TYPE ST_HMI_SAFETY_IN :
STRUCT
	bQuitSafety,
	
	bQuitAreaST10,
	bUnlockDoorST33	: BOOL;
END_STRUCT
END_TYPE

(* stored: Version 1.1.0.1, ProductVersion 3.1.4024.12
   DUT ST_HMI_SAFETY_IN: Id {ab1ef7de-b48d-4de3-b101-a0e09ef21d9b} *)
